(* PLC project  *)

PROGRAM P
  VAR  (* added by the conversion: wires and edge detectors of the diagram *)
    _AND3_OUT : BOOL;
  END_VAR

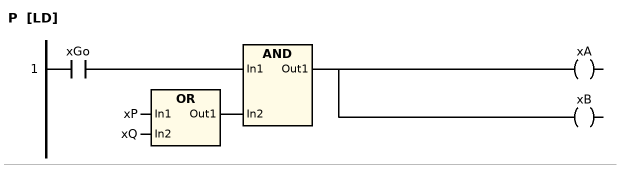
(* LD diagram, written out as Structured Text *)
_AND3_OUT := xGo AND (xP OR xQ);
xA := _AND3_OUT;
xB := _AND3_OUT;
END_PROGRAM
